// TIA Portal V17 export
// export: Created 2024-09-03T21:55:05.9609969Z, ExportSetting WithDefaults, DisplayName Totally Integrated Automation Portal, DisplayVersion V17 Update 7, DisplayName TIA Portal Openness, DisplayVersion V17 Update 7, DisplayName TIA Portal Version Control Interface, DisplayVersion V17, DisplayName SINAMICS Startdrive Advanced, DisplayVersion V17 SP2, DisplayName SINAMICS Startdrive G110M, G120, G120C, G120D, G120P, G115D, DisplayVersion V17 SP2, DisplayName SINAMICS Startdrive G130, G150, S120, S150, SINAMICS MV, S210, DisplayVersion V17 SP2, DisplayName STEP 7 Professional, DisplayVersion V17 Update 7, DisplayName STEP 7 Safety, DisplayVersion V17 Update 6, DisplayName WinCC Advanced / Unified PC, DisplayVersion V17 Update 7
TYPE "udtModes"
// stored: IsFailsafeCompliant false
   STRUCT
      activeMode : Int;
      switch : Struct
         auto : Bool;
         poloautomaActivated : Bool;
         stepModeActivated : Bool;
      END_STRUCT;
      button : Struct
         basic : Struct
            request : Struct
               button : Bool;
               visibility : Bool;
            END_STRUCT;
         END_STRUCT;
         auto : Struct
            startRequest : Struct
               button : Bool;
               visibility : Bool;
            END_STRUCT;
            stopRequest : Struct
               button : Bool;
               visibility : Bool;
            END_STRUCT;
            emptyRequest : Struct
               button : Bool;
               visibility : Bool;
            END_STRUCT;
         END_STRUCT;
         "step" : Bool;
         poloautomatStart : Array[0..25] of Bool;
      END_STRUCT;
      modeChanged : Bool;
      autoStatus : Struct
         stopping : Bool;
         stopped : Bool;
         emptying : Bool;
         empty : Bool;
      END_STRUCT;
      StationNrForPoloautomat_step : Int;
   END_STRUCT;
END_TYPE
